// SIMATIC STEP 7 (V5.x) project Печь BLEMA
// CPU: CPU 312
// station: Hardware
// station: SIMATIC 300(1)
// station: P_ADR_BUS
// program: S7 Program(1)

SYMBOL_TABLE
"FC1"	FC 1	FC 1
"S3.6"	I 4.0	BOOL	// Сброс
"S0.1-S0.2"	I 4.1	BOOL	// Общий СТОП
"S4.1"	I 4.2	BOOL	// Переключатель РУЧНОЕ-АВТОМАТ
"S3.1"	I 4.3	BOOL	// ПУСК транспортеров
"S3.2"	I 4.4	BOOL	// СТОП транспортеров
"S3.3"	I 4.5	BOOL	// ПУСК горелок
"S3.4"	I 4.6	BOOL	// СТОП горелок
"K7.1-K7.2"	I 5.0	BOOL	// Контроль пламени горелок 1,2
"K7.3-K7.4"	I 5.1	BOOL	// Контроль пламени горелок 3,4
"B1.1-B1.4"	I 5.2	BOOL	// Контроль первичного воздуха на горелках
"AB1"	I 5.3	BOOL	// Автомат защиты М2.1
"AB2"	I 5.4	BOOL	// Автомат защиты М2.2
"AB3"	I 5.5	BOOL	// Автомат защиты М2.3
"AB9"	I 5.6	BOOL	// Автомат защиты М2.10
"U1"	I 8.0	BOOL	// Контроль работы ЧП1
"U2"	I 8.1	BOOL	// Контроль работы ЧП2
"U3"	I 8.2	BOOL	// Контроль работы ЧП3
"U4"	I 8.3	BOOL	// Контроль работы ЧП4
"U5"	I 8.4	BOOL	// Контроль работы ЧП5
"U6"	I 8.5	BOOL	// Контроль работы ЧП6
"m1.0"	M 1.0	BOOL	// СТОП транспортеров печи
"m1.1"	M 1.1	BOOL	// ПУСК транспортеров печи
"m1.2"	M 1.2	BOOL	// Контроль работы транспортеров печи
"M2.4"	Q 12.0	BOOL	// Транспортер №1 перед печью
"M2.5-M2.6"	Q 12.1	BOOL	// Транспортеры №2 и №3 печи
"M2.7"	Q 12.2	BOOL	// Поворот на печи
"M2.8"	Q 12.3	BOOL	// Транспортер №4 после печи
"M2.9"	Q 12.4	BOOL	// Подъемник и верхний транспортер (цепь 1)
"M2.11"	Q 12.5	BOOL	// Верхний транспортер (цепь 2)
"K9.1"	Q 16.0	BOOL	// Воздушный компрессор
"K9.2"	Q 16.1	BOOL	// Вунтилятор вторичного воздуха
"K9.3"	Q 16.2	BOOL	// Водяной насос
"K9.4"	Q 16.3	BOOL	// Поворот на верхнем транспортере
"H1.3"	Q 16.4	BOOL	// Помеха
"H1.4"	Q 16.5	BOOL	// РАБОТА печь 1,2
"H1.5"	Q 16.6	BOOL	// РАБОТА печь 3,4
"Y1.3"	Q 20.0	BOOL	// Общий газ горелки 1,2
"Y1.4"	Q 20.1	BOOL	// Общий газ горелки 3,4
"Y1.5"	Q 20.2	BOOL	// Рабочий газ горелки 1,2
"Y1.6"	Q 20.3	BOOL	// Рабочий газ горелки 3,4
"Y1.7"	Q 20.4	BOOL	// Зажигающий газ горелки 1,2
"Y1.8"	Q 20.5	BOOL	// Зажигающий газ горелки 3,4
"Y1.9"	Q 20.6	BOOL	// Первичный воздух горелок 1,2
"Y1.10"	Q 20.7	BOOL	// Первичный воздух горелок 3,4
"Y1.11"	Q 24.0	BOOL	// Выброс банки
"Y2.1"	Q 24.1	BOOL	// Воздушная заслонка вторичного воздуха
"t1"	T 1	TIMER	// Таймер задержки закрытия заслонки
"t2"	T 2	TIMER	// Таймер открытия заслонки
"t3"	T 3	TIMER	// Таймер включения электроподжига
END_SYMBOL_TABLE

FUNCTION "FC1" : VOID	// FC 1
VERSION : 0.1
BEGIN
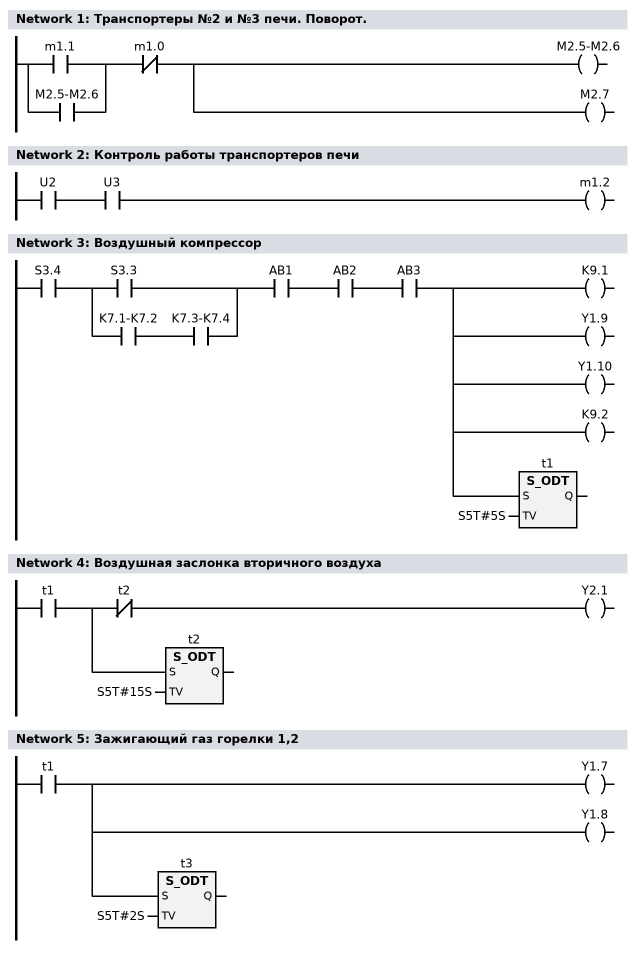
NETWORK
TITLE = Транспортеры №2 и №3 печи. Поворот.
      A(;
      O     "m1.1";
      O     "M2.5-M2.6";
      );
      AN    "m1.0";
      =     "M2.5-M2.6";
      =     "M2.7";
NETWORK
TITLE = Контроль работы транспортеров печи
      A     "U2";
      A     "U3";
      =     "m1.2";
NETWORK
TITLE = Воздушный компрессор
      A     "S3.4";
      A(;
      O     "S3.3";
      O;
      A     "K7.1-K7.2";
      A     "K7.3-K7.4";
      );
      A     "AB1";
      A     "AB2";
      A     "AB3";
      =     L 0.0;
      A     L 0.0;
      BLD   102;
      =     "K9.1";
      A     L 0.0;
      BLD   102;
      =     "Y1.9";
      A     L 0.0;
      BLD   102;
      =     "Y1.10";
      A     L 0.0;
      BLD   102;
      =     "K9.2";
      A     L 0.0;
      L     S5T#5S;
      SD    "t1";
      NOP   0;
      NOP   0;
      NOP   0;
      NOP   0;
NETWORK
TITLE = Воздушная заслонка вторичного воздуха
      A     "t1";
      =     L 0.0;
      A     L 0.0;
      AN    "t2";
      =     "Y2.1";
      A     L 0.0;
      L     S5T#15S;
      SD    "t2";
      NOP   0;
      NOP   0;
      NOP   0;
      NOP   0;
NETWORK
TITLE = Зажигающий газ горелки 1,2
      A     "t1";
      =     L 0.0;
      A     L 0.0;
      BLD   102;
      =     "Y1.7";
      A     L 0.0;
      BLD   102;
      =     "Y1.8";
      A     L 0.0;
      L     S5T#2S;
      SD    "t3";
      NOP   0;
      NOP   0;
      NOP   0;
      NOP   0;
END_FUNCTION

ORGANIZATION_BLOCK OB 1
TITLE = "Main Program Sweep (Cycle)"
VERSION : 0.1
VAR_TEMP
  OB1_EV_CLASS : BYTE ;	//Bits 0-3 = 1 (Coming event), Bits 4-7 = 1 (Event class 1)
  OB1_SCAN_1 : BYTE ;	//1 (Cold restart scan 1 of OB 1), 3 (Scan 2-n of OB 1)
  OB1_PRIORITY : BYTE ;	//Priority of OB Execution
  OB1_OB_NUMBR : BYTE ;	//1 (Organization block 1, OB1)
  OB1_RESERVED_1 : BYTE ;	//Reserved for system
  OB1_RESERVED_2 : BYTE ;	//Reserved for system
  OB1_PREV_CYCLE : INT ;	//Cycle time of previous OB1 scan (milliseconds)
  OB1_MIN_CYCLE : INT ;	//Minimum cycle time of OB1 (milliseconds)
  OB1_MAX_CYCLE : INT ;	//Maximum cycle time of OB1 (milliseconds)
  OB1_DATE_TIME : DATE_AND_TIME ;	//Date and time OB1 started
END_VAR
BEGIN
// (block stored without names or comments; labels and parameter names are numbered)
END_ORGANIZATION_BLOCK
